(* Schneider Machine Expert - Basic project Motor_Incremental_Test, file version 3.0.0.0 *)
(* ProjectInformations: Name=New project *)

HARDWARE
  Cpu 0: TM221CE16T
  ModuleExtensionObject 0: TM3DI32K
  ModuleExtensionObject 1: TM3DQ32TK
  ModuleExtensionObject 2: TM3AI8/G
  ModuleExtensionObject 3: TM3TI4D/G
  ModuleExtensionObject 4: TM3TI4/G
  Cartridge1 0: TMC2AI2
  Cartridge2 0: TMC2TI2
  EthernetConfiguration: NetworkName=M221, IpAllocationMode=FixedAddress, IpAddress=0.0.0.0, SubnetMask=0.0.0.0
  EthernetConfiguration: NetworkName=M221, IpAllocationMode=FixedAddress, IpAddress=0.0.0.0, SubnetMask=0.0.0.0
  EthernetConfiguration: NetworkName=M221, IpAllocationMode=FixedAddress, IpAddress=0.0.0.0, SubnetMask=0.0.0.0
  SerialLineConfiguration: Baud=Baud19200, Parity=ParityEven, DataBits=DataBits8, StopBits=StopBits1, PhysicalMedium=PhysicalMediumRs485, TransmissionMode=TransmissionModeModbusRtu, SlaveId=1, Addressing=SlaveAddressing
  MastTask: UsePeriodScanMode=false, PeriodScan=100
  FastTask: Period=255
  CpuBehavior: StartingMode=StartAsPreviousState, AutoSaveRamOnEeprom=true, WatchdogPeriod=250

SYMBOLS  (address, symbol, comment, settings)
  %M0       SYSTEM_READY
  %S0       SB_COLDSTART  "Indicates or executes a cold start (data initialized to default values)"
  %S1       SB_WARMSTART  "Indicates there was a warm start with data backup"
  %TM0        [Preset=3, Base=OneSecond]
  %I0.0     EMERGENCY_PB

POU New POU
  (* SectionNumber=0 *)

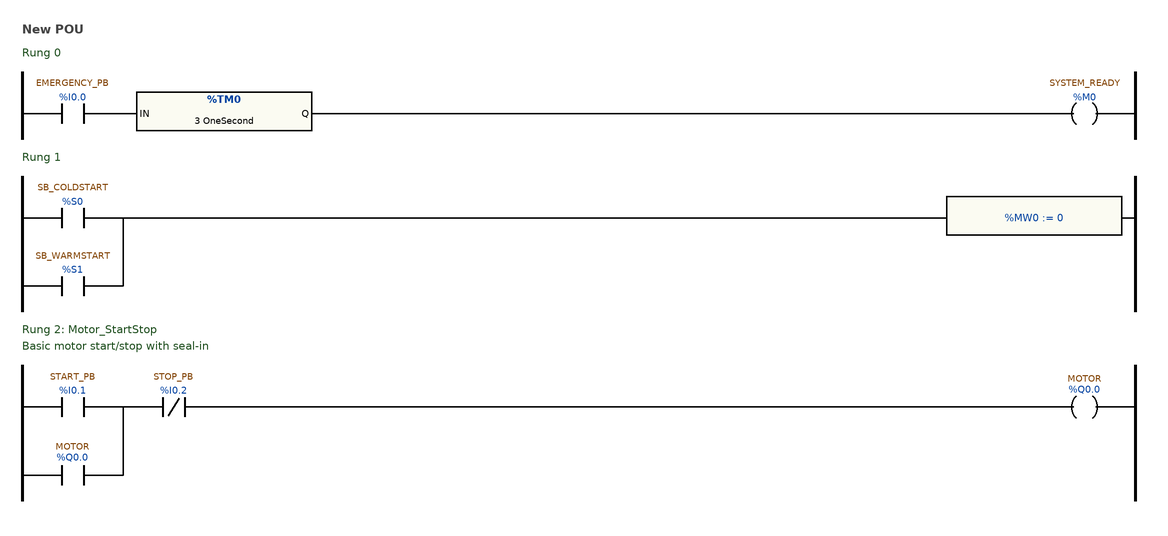

// Rung 0
  BLK %TM0
  LD %I0.0                (* EMERGENCY_PB *)
  IN
  OUT_BLK
  LD Q
  ST %M0                  (* SYSTEM_READY *)
  END_BLK
  // as ST:
  //   %TM0(IN := EMERGENCY_PB);
  //   SYSTEM_READY := %TM0.Q;

// Rung 1
  LD %S0                  (* SB_COLDSTART *)
  OR %S1                  (* SB_WARMSTART *)
  [ %MW0 := 0 ]
  // as ST:
  //   IF SB_COLDSTART OR SB_WARMSTART THEN %MW0 := 0; END_IF;

// Rung 2: Motor_StartStop
// Basic motor start/stop with seal-in
  LD %I0.1                (* Start *)
  OR %Q0.0                (* Seal-in *)
  ANDN %I0.2              (* Stop *)
  ST %Q0.0                (* Motor *)
  // %I0.1: Start Button
  // %I0.2: Stop Button NC
  // %Q0.0: Motor Output
  // %Q0.0: Seal-in
  // as ST:
  //   %Q0.0 := (%I0.1 OR %Q0.0) AND NOT %I0.2;
